Universal Robots PolyScope program: RC_E8_PLACE_830.urp

Program RC_E8_PLACE_830 (createdIn=3.0.0 lastSavedIn=3.0.0 directory=/programs installation=default)
Robot Program (runOnlyOnce=true motionType=MoveJ speed=1.047198 acceleration=1.396263 useActiveTCP=false)
  'Program generated by RoboDK v4.1.0 for UR3e_HORNO on 06/09/2022 17:08:19'
  'Using nominal kinematics.'
  'Using Ref. Frame Traslado C: p[0.369000, -0.220000, 0.032000, 0.000000, 0.000000, 0.000000]'
  'Using TCP 0208-0001-0001-307-000-3 Horno: p[0.000000, 0.000000, 0.164750, 0.000000, 0.000000, 0.000000]'
  Script: set_tcp(p[0.000000, 0.000000, 0.164750, 0.000000, 0.000000, 0.000000])
  Script: movej([0.453224, -1.802935, -0.994995, -3.455038, 0.479382, 3.143909],0.60000,0.12500,0,0.0000)
  MoveL speed 100 mm/s, acceleration 120 mm/s^2 (useActiveTCP=true)
    Waypoint Waypoint_1: TCP in base x=644.953 y=-490 z=179 mm, rx=-0.0414 ry=-2.2292 rz=2.1985 rad; joints [24.906, -111.557, -110.388, -136.249, 26.405, 179.024] deg; flange x=649.231 y=-325.322 z=181.308 mm, rx=-0.0414 ry=-2.2292 rz=2.1985 rad
  'Detach from 0208-0001-0001-307-000-3 Horno'
  Script: movej([0.453224, -1.802935, -0.994995, -3.455038, 0.479382, 3.143909],0.12000,0.10000,0,0.0000)
